(* CODESYS project i2cTeste.project

Project tree, tasks and I/O mapping:
  Device : CODESYS Control for Raspberry Pi SL, 3S - Smart Software Solutions GmbH, version 3.5.16.0
    application Application
      libraries: Standard, * (System); VisuDialogs, * (System)
      task ENIPScannerServiceTask (cyclic, interval 500 ms, priority 30) calls EtherNet_IP_Scanner.ServiceCycle
      task MainTask (cyclic, interval 50 ms, priority 1) calls PLC_PRG
      task ENIPScannerIOTask (cyclic, interval 20 ms, priority 1) calls EtherNet_IP_Scanner.IOCycle
      task VISU_TASK (cyclic, interval 100 ms, priority 31) calls VisuElems.Visu_Prg
      global variables IO
      visualisation Start
      global variables GVL
      program PLC_PRG [ST]
    Onewire
    Camera device
      <Empty>
    I²C
      I2C_master : I2C master, 3S - Smart Software Solutions GmbH, version 1.0.0.0
        I2C_Encoder_Emulator : I2C Encoder Emulator, Open Source, version 1.0.0.0
            settings: I2C Address = 8
            unmapped channels: Command, RPM, Resolucao Encoder
    SoftMotion General Axis Pool
    GPIOs_A_B : GPIOs B+/Pi2, 3S - Smart Software Solutions GmbH, version 3.5.16.0
        unmapped channels: digital inputs (GPIO0..GPIO31), digital outputs (GPIO0..GPIO31)
    Ethernet : Ethernet, 3S - Smart Software Solutions GmbH, version 3.5.16.0
        settings: IPAddress = [192,168,1,10]; SubnetMask = [255,255,255,0]; GatewayAddress = [192,168,1,1]; NetworkInterfaceName = 'eth0'; NetworkInterfaceName = "eth0"; SaveCommunicationSettings = FALSE
      EtherNet_IP_Scanner : EtherNet/IP Scanner, 3S - Smart Software Solutions GmbH, order no. 1, version 3.5.16.0
        UR20_FBC_EIP : UR20-FBC-EIP, Weidmueller Interface, order no. 1334920000, version Major Revision=16#1, Minor Revision = 16#3
            settings: INITIALIZED = TRUE; IP address of Target = [16#C0,16#A8,16#01,16#CA]; Keying.Check Major Revision = FALSE; Keying.Check Minor Revision = FALSE; RequiredConfigVersion = 50660864; Number of Connections = 1; Connection Settings.Requested packet intervall (µs) = 20000; Connection Settings.OT Connection Parameters = 18442; Connection Settings.TO Connection Parameters = 18438; Connection Settings.Connection Flags = 1056; Connection Settings.Connection Path Size = 8; Connection Path = [16#20,16#04,16#24,16#01,16#2C,16#66,16#2C,16#65]; Status register.ReadOnly = False; Status register.BitSize = 16; Status register.DataSize = 2; Input Process DataParam1.ReadOnly = False; Input Process DataParam1.BitSize = 8; Input Process DataParam1.DataSize = 1; Input Process DataParam2.ReadOnly = False; Input Process DataParam2.BitSize = 8; Input Process DataParam2.DataSize = 1; Control Register.ReadOnly = False; Control Register.BitSize = 16; Control Register.DataSize = 2; Output Process DataParam1.ReadOnly = False; Output Process DataParam1.BitSize = 8; Output Process DataParam1.DataSize = 1; Output Process DataParam2.ReadOnly = False; Output Process DataParam2.BitSize = 8; Output Process DataParam2.DataSize = 1; Status register.Name = 'Status register'; Status register.HelpString = ''; Status register.ReadOnly = False; Status register.BitSize = 16; Status register.DataSize = 2; Status register.DataType = 'WORD'; Input Process DataParam1.Name = 'Input Process DataParam1'; Input Process DataParam1.HelpString = ''; Input Process DataParam1.ReadOnly = False; Input Process DataParam1.BitSize = 8;
              Input Process DataParam1.DataSize = 1; Input Process DataParam1.DataType = 'BYTE'; Input Process DataParam2.Name = 'Input Process DataParam2'; Input Process DataParam2.HelpString = ''; Input Process DataParam2.ReadOnly = False; Input Process DataParam2.BitSize = 8; Input Process DataParam2.DataSize = 1; Input Process DataParam2.DataType = 'BYTE'; Control Register.Name = 'Control Register'; Control Register.HelpString = ''; Control Register.ReadOnly = False; Control Register.BitSize = 16; Control Register.DataSize = 2; Control Register.DataType = 'WORD'; Output Process DataParam1.Name = 'Output Process DataParam1'; Output Process DataParam1.HelpString = ''; Output Process DataParam1.ReadOnly = False; Output Process DataParam1.BitSize = 8; Output Process DataParam1.DataSize = 1; Output Process DataParam1.DataType = 'BYTE'; Output Process DataParam2.Name = 'Output Process DataParam2'; Output Process DataParam2.HelpString = ''; Output Process DataParam2.ReadOnly = False; Output Process DataParam2.BitSize = 8; Output Process DataParam2.DataSize = 1; Output Process DataParam2.DataType = 'BYTE'; ConfigVersion = 50660864
            unmapped channels: Status register, Input Process DataParam1, Input Process DataParam2, Control Register, Output Process DataParam1, Output Process DataParam2
    SPI
  libraries: VisuSymbols, 3.5.10.0 (System)
  Recursos/
    function block PULSE [ST]
  text list GlobalTextList
*)

// Device/Application/IO
{attribute 'qualified_only'}
VAR_GLOBAL
	GPIO_DI_04	AT %IX32.4	: BOOL;
	GPIO_DI_17	AT %IX34.1	: BOOL;
	GPIO_DI_18	AT %IX34.2	: BOOL;
	GPIO_DI_22	AT %IX34.6	: BOOL;
	GPIO_DI_23	AT %IX34.7	: BOOL;
	GPIO_DI_24	AT %IX35.0	: BOOL;
	GPIO_DI_25	AT %IX35.1	: BOOL;
	GPIO_DI_27	AT %IX35.3	: BOOL;
	GPIO_DI_28	AT %IX35.4	: BOOL;
	GPIO_DI_29	AT %IX35.5	: BOOL;
	GPIO_DI_30	AT %IX35.6	: BOOL;
	GPIO_DI_31	AT %IX35.7	: BOOL;

	GPIO_DO_04	AT %QX8.4	: BOOL;
	GPIO_DO_17	AT %QX10.1	: BOOL;
	GPIO_DO_18	AT %QX10.2	: BOOL;
	GPIO_DO_22	AT %QX10.6	: BOOL;
	GPIO_DO_23	AT %QX10.7	: BOOL;
	GPIO_DO_24	AT %QX11.0	: BOOL;
	GPIO_DO_25	AT %QX11.1	: BOOL;
	GPIO_DO_27	AT %QX11.3	: BOOL;
	GPIO_DO_28	AT %QX11.4	: BOOL;
	GPIO_DO_29	AT %QX11.5	: BOOL;
	GPIO_DO_30	AT %QX11.6	: BOOL;
	GPIO_DO_31	AT %QX11.7	: BOOL;
	

	REM_DI01	AT %IX2.0	: BOOL;
	REM_DI02	AT %IX2.1	: BOOL;
	REM_DI03	AT %IX2.2	: BOOL;
	REM_DI04	AT %IX2.3	: BOOL;
	REM_DI05	AT %IX2.4	: BOOL;
	REM_DI06	AT %IX2.5	: BOOL;
	REM_DI07	AT %IX2.6	: BOOL;
	REM_DI08	AT %IX2.7	: BOOL;
	REM_DI09	AT %IX3.0	: BOOL;
	REM_DI10	AT %IX3.1	: BOOL;
	REM_DI11	AT %IX3.2	: BOOL;
	REM_DI12	AT %IX3.3	: BOOL;
	REM_DI13	AT %IX3.4	: BOOL;
	REM_DI14	AT %IX3.5	: BOOL;
	REM_DI15	AT %IX3.6	: BOOL;
	REM_DI16	AT %IX3.7	: BOOL;
	
	REM_DO01	AT %QX2.0	: BOOL;
	REM_DO02	AT %QX2.1	: BOOL;
	REM_DO03	AT %QX2.2	: BOOL;
	REM_DO04	AT %QX2.3	: BOOL;
	REM_DO05	AT %QX2.4	: BOOL;
	REM_DO06	AT %QX2.5	: BOOL;
	REM_DO07	AT %QX2.6	: BOOL;
	REM_DO08	AT %QX2.7	: BOOL;
	REM_DO09	AT %QX3.0	: BOOL;
	REM_DO10	AT %QX3.1	: BOOL;
	REM_DO11	AT %QX3.2	: BOOL;
	REM_DO12	AT %QX3.3	: BOOL;
	REM_DO13	AT %QX3.4	: BOOL;
	REM_DO14	AT %QX3.5	: BOOL;
	REM_DO15	AT %QX3.6	: BOOL;
	REM_DO16	AT %QX3.7	: BOOL;
	
END_VAR

// Device/Application/GVL
//{attribute 'qualified_only'}
VAR_GLOBAL
	PI	: REAL := 3.141592;
END_VAR

// Device/Application/PLC_PRG
PROGRAM PLC_PRG
VAR
	cmdAvancar	: BOOL;
	cmdRecuar	: BOOL;
	rpm	: INT;
	resolucao	: INT:= 1024;
	upAvancar	: R_Trig;
	upRecuar	: R_Trig;	
	tPeriodoCiclo	: DWORD;
	tFase	: DWORD;
END_VAR

upAvancar(CLK:= cmdAvancar);
IF upAvancar.Q THEN
	cmdRecuar:= FALSE;
END_IF

upRecuar(CLK:= cmdRecuar);
IF upRecuar.Q THEN
	cmdAvancar:= FALSE;
END_IF

IF cmdAvancar THEN
	I2C_Encoder_Emulator.cmd:= 1;
ELSIF cmdRecuar THEN
	I2C_Encoder_Emulator.cmd:= 2;
ELSE	
	I2C_Encoder_Emulator.cmd:= 0;
END_IF

I2C_Encoder_Emulator.rpm:= rpm;
I2C_Encoder_Emulator.resolucao:= resolucao;

IF rpm <> 0 AND resolucao <> 0 THEN
	tFase:= (60000000 / rpm) / resolucao;
	tPeriodoCiclo:= tFase * 4;
END_IF;

END_PROGRAM

// Recursos/PULSE
FUNCTION_BLOCK PULSE
VAR_INPUT
	EN	: BOOL;
	IN	: BOOL;
	PT_HIGH	: TIME;
	PT_LOW	: TIME;
END_VAR
VAR_OUTPUT
	Q	: BOOL;
	END	: BOOL;
	ET_HIGH	: TIME;
	ET_LOW	: TIME;
	RT_HIGH	: TIME;
	RT_LOW	: TIME;
END_VAR
VAR
	TIME_old	: TIME;
	EN_old	: BOOL;
END_VAR

IF PT_HIGH > T#49D17H2M THEN PT_HIGH:= T#49D17H2M;	END_IF
IF PT_LOW > T#49d17h2m THEN PT_LOW:= T#49d17h2m;	END_IF

IF IN THEN
	IF EN THEN
		IF EN_old < EN THEN
			TIME_old:= TIME();
			EN_old:= EN;
		ELSE

			IF ET_HIGH < PT_HIGH THEN
				Q:= TRUE;
			ELSIF ET_LOW < PT_LOW THEN
				Q:= FALSE;
			ELSE
				ET_HIGH:= T#0s;
				ET_LOW:= T#0s;
				TIME_old:= TIME();
			END_IF

			IF TIME() > TIME_old AND ET_HIGH <= T#49d17h2m AND ET_LOW <= T#49d17h2m THEN
				IF Q THEN
					ET_HIGH:= ET_HIGH + (TIME() - TIME_old);
				ELSE
					ET_LOW:= ET_LOW + (TIME() - TIME_old);
				END_IF
				TIME_old:= TIME();
			END_IF
		END_IF
	ELSE
		EN_old:=FALSE;
	END_IF

ELSE
	EN_old:= FALSE;
	ET_HIGH:= t#0s;
	ET_LOW:= t#0s;
	Q:= FALSE;
END_IF

IF PT_HIGH > ET_HIGH THEN
	RT_HIGH:= PT_HIGH - ET_HIGH;
ELSE
	RT_HIGH:= T#0s;
END_IF

IF PT_LOW > ET_LOW THEN
	RT_LOW:= PT_LOW - ET_LOW;
ELSE
	RT_LOW:= T#0s;
END_IF

END_FUNCTION_BLOCK

// Device/Application/Start
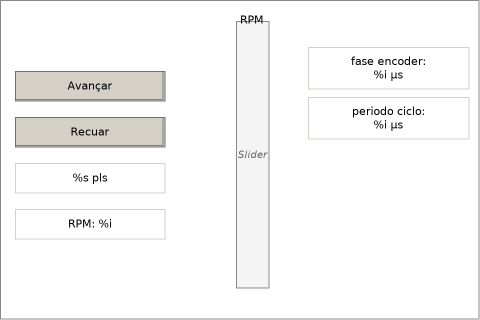
VISUALIZATION Start  // 480x320
    Button (15,71 150x30), "Avançar"
        toggle PLC_PRG.cmdAvancar
    Button (15,117 150x30), "Recuar"
        toggle PLC_PRG.cmdRecuar
    Slider (236,21 33x267), variable: PLC_PRG.rpm, scale 0..2000
    Textfield (15,163 150x30), "%s pls", text variable: PLC_PRG.resolucao
        OnMouseUp: write the text variable via Default
    Textfield (15,209 150x30), "RPM: %i", text variable: PLC_PRG.rpm
    Textfield (308,47 161x42), "fase encoder: %i µs", text variable: PLC_PRG.tFase
    Label (228,5 48x30), "RPM"
    Textfield (308,97 161x42), "periodo ciclo: %i µs", text variable: PLC_PRG.tPeriodoCiclo
END_VISUALIZATION
